TYPE SyncUnitInfoData :
STRUCT
	{attribute addProperty Name "ObjectId"}
	ObjectId AT %I* : OTCID;
	{attribute addProperty Name "State"}
    State AT %I* : UINT;
	{attribute addProperty Name "SlaveCount"}
    SlaveCount AT %I* : UINT;
END_STRUCT
END_TYPE

(* stored: Version 1.1.0.1, ProductVersion 3.1.4024.9
   DUT SyncUnitInfoData: Id {195d10da-9e0b-0061-2728-7a4c719162f6} *)
